(* PLC project Tc3_EventLogger.FB_TcAlarm.Create Demo, tc3-libraries-kb TwinCAT 3.1 *)
(* stored: creationDateTime 2026-05-11T01:00:00, modificationDateTime 2026-05-11T01:00:00 *)

PROGRAM P_Demo_FB_TcAlarm_Create
  VAR
    fbTcAlarm : FB_TcAlarm;  (* Tc3_EventLogger.FB_TcAlarm 实例 *)
    arg_eventClass : GUID;  (* VAR_INPUT eventClass *)
    arg_nEventId : UDINT;  (* VAR_INPUT nEventId *)
    arg_eSeverity : TcEventSeverity;  (* VAR_INPUT eSeverity *)
    arg_bWithConfirmation : BOOL;  (* VAR_INPUT bWithConfirmation *)
    arg_ipSourceInfo : I_TcSourceInfo;  (* VAR_INPUT ipSourceInfo *)
    hr : HRESULT;  (* 返回值 HRESULT *)
  END_VAR

            // ============================================================
// Tc3_EventLogger.FB_TcAlarm.Create 演示程序（OO 方法）
// ============================================================
// 验证步骤：
//   1. 引用 Tc3_EventLogger（及依赖类型所在库 Tc2_System 等）
//   2. 编译 + 登录
//   3. 在线给 arg_* 赋值（eventClass、nEventId、eSeverity、bWithConfirmation、ipSourceInfo）
//   4. 触发 Create，监视返回的 hr（S_OK 表示成功）
// ============================================================

hr := fbTcAlarm.Create(
    eventClass := arg_eventClass,
    nEventId := arg_nEventId,
    eSeverity := arg_eSeverity,
    bWithConfirmation := arg_bWithConfirmation,
    ipSourceInfo := arg_ipSourceInfo
);

          
END_PROGRAM
